KUKA KRL program: ho_60101.src, ho_60101.dat

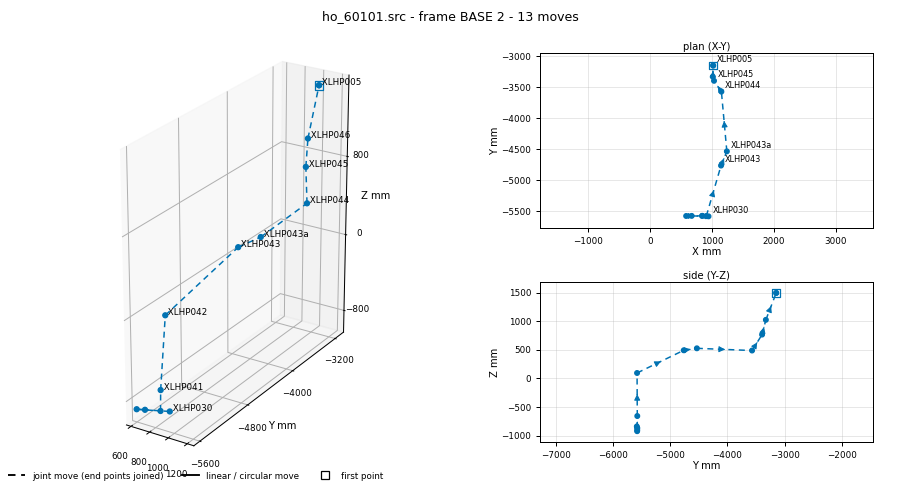
[picture p0: tool path of ho_60101.src in frame BASE 2, 13 of 19 moves have a stored position in this frame; points joined in program order, loops and branches not executed]
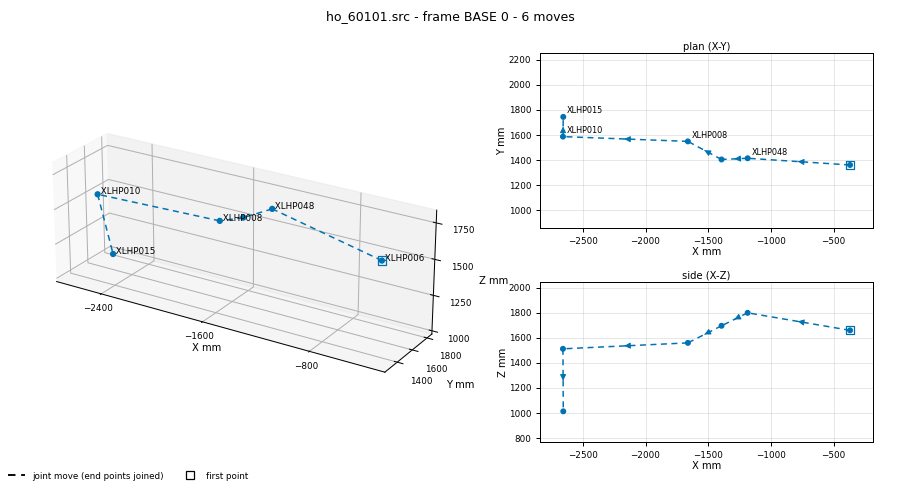
[picture p1: tool path of ho_60101.src in frame BASE 0, 6 of 19 moves have a stored position in this frame; points joined in program order, loops and branches not executed]
--- ho_60101.src ---
&ACCESS RVO2
&REL 599
&COMMENT Pega Lateral
&PARAM DISKPATH = KRC:\R1\Program\MANIPULACAO LTC
DEF ho_60101( )
;FOLD INI
   ;FOLD BASISTECH INI
      GLOBAL INTERRUPT DECL 3 WHEN $STOPMESS==TRUE DO IR_STOPM ( )
      INTERRUPT ON 3
      BAS (#INITMOV,0 )
   ;ENDFOLD (BASISTECH INI)
   ;FOLD SPOTTECH INI
      USERSPOT(#INIT)
   ;ENDFOLD (SPOTTECH INI)
   ;FOLD GRIPPERTECH INI
      USER_GRP(0,DUMMY,DUMMY,GDEFAULT)
   ;ENDFOLD (GRIPPERTECH INI)
   ;FOLD USER INI
      ;Make your modifications here

   ;ENDFOLD (USER INI)
;ENDFOLD (INI)

; Estacao P13.060 - Robo R1
; Programa: Pega da Lateral Accelo (GRIPPER)
; Caracterização dos meios de produção:
; 02/09/2014 09:15 Changes by KUKA Roboter do Brasil

chk_w2_wechs_ok ( )           ; CHECK FERRAMENTA: GRIPPER

;FOLD Kollision.Ueberwachung_3_Ein ;%{PE}%MKUKATPUSER
COLLSTOP( 3, 1 ) ;INTERRUPTUEBERWACHT
;ENDFOLD

;FOLD PTP LHP005  Vel=50 % PDAT23 Tool[2] Base[2];%{PE}%R 4.1.15,%MKUKATPBASIS,%CMOVE,%VPTP,%P 1:PTP, 2:LHP005, 3:, 5:50, 7:PDAT23
$BWDSTART=FALSE
PDAT_ACT=PPDAT23
BAS (#PTP_DAT )
FDAT_ACT=FLHP005
BAS (#FRAMES )
BAS (#VEL_PTP,50 )
PTP  XLHP005
;ENDFOLD
;FOLD PTP LHP006 Vel=100 % PDAT1 Tool[2]:Gripper Lat Esq Accelo Base[0];%{PE}%R 8.2.20,%MKUKATPBASIS,%CMOVE,%VPTP,%P 1:PTP, 2:LHP006, 3:, 5:100, 7:PDAT1
$BWDSTART=FALSE
PDAT_ACT=PPDAT1
FDAT_ACT=FLHP006
BAS(#PTP_PARAMS,100)
PTP XLHP006
;ENDFOLD

;FOLD SET GRP 1  State= OPN  GDAT7;%{PE}%R 4.1.7,%MKUKATPGRP,%CGRP,%VGRP,%P 2:1, 4:1, 5:#NO, 6:GDAT7, 8:0, 10:0
H50(GRP,1,1,GGDAT7)
;ENDFOLD
chk_grp1_opn ( )

;FOLD OUT 3351 'R1_Busca Peca Accelo' State=TRUE ;%{PE}%R 8.2.20,%MKUKATPBASIS,%COUT,%VOUTX,%P 2:3351, 3:R1_Busca Peca Accelo, 5:TRUE, 6:
$OUT[3351]=TRUE
;ENDFOLD
;FOLD OUT 3361 'R1_Solicita Lib. Entrar EST 060EL_621' State=TRUE ;%{PE}%R 8.2.20,%MKUKATPBASIS,%COUT,%VOUTX,%P 2:3361, 3:R1_Solicita Lib. Entrar EST 060EL_621, 5:TRUE, 6:
$OUT[3361]=TRUE
;ENDFOLD
;FOLD WAIT FOR ( IN 3351 'R1_Aguarda Lib. Buscar Lat. Accelo' );%{PE}%R 8.2.20,%MKUKATPBASIS,%CEXT_WAIT_FOR,%VEXT_WAIT_FOR,%P 2:, 4:, 5:$IN, 6:3351, 7:R1_Aguarda Lib. Buscar Lat. Accelo, 9:
WAIT FOR  ( $IN[3351] )
;ENDFOLD
;FOLD OUT 3351 'R1_Busca Peca Accelo' State=FALSE ;%{PE}%R 8.2.20,%MKUKATPBASIS,%COUT,%VOUTX,%P 2:3351, 3:R1_Busca Peca Accelo, 5:FALSE, 6:
$OUT[3351]=FALSE
;ENDFOLD
;FOLD OUT 3361 'R1_Solicita Lib. Entrar EST 060EL_621' State=FALSE ;%{PE}%R 8.2.20,%MKUKATPBASIS,%COUT,%VOUTX,%P 2:3361, 3:R1_Solicita Lib. Entrar EST 060EL_621, 5:FALSE, 6:
$OUT[3361]=FALSE
;ENDFOLD
;FOLD OUT 3367 'R1_Solda Respot Geo1 OK' State=FALSE ;%{PE}%R 8.2.20,%MKUKATPBASIS,%COUT,%VOUTX,%P 2:3367, 3:R1_Solda Respot Geo1 OK, 5:FALSE, 6:
$OUT[3367]=FALSE
;ENDFOLD

;FOLD PTP LHP048 CONT Vel=100 % PDAT12 Tool[2]:Gripper Lat Esq Accelo Base[0];%{PE}%R 8.2.20,%MKUKATPBASIS,%CMOVE,%VPTP,%P 1:PTP, 2:LHP048, 3:C_DIS, 5:100, 7:PDAT12
$BWDSTART=FALSE
PDAT_ACT=PPDAT12
FDAT_ACT=FLHP048
BAS(#PTP_PARAMS,100)
PTP XLHP048 C_DIS
;ENDFOLD
;FOLD PTP LHP007 CONT Vel=100 % PDAT11 Tool[2]:Gripper Lat Esq Accelo Base[0];%{PE}%R 8.2.20,%MKUKATPBASIS,%CMOVE,%VPTP,%P 1:PTP, 2:LHP007, 3:C_DIS, 5:100, 7:PDAT11
$BWDSTART=FALSE
PDAT_ACT=PPDAT11
FDAT_ACT=FLHP007
BAS(#PTP_PARAMS,100)
PTP XLHP007 C_DIS
;ENDFOLD
;FOLD PTP LHP008 CONT Vel=100 % PDAT13 Tool[2]:Gripper Lat Esq Accelo Base[0];%{PE}%R 8.2.20,%MKUKATPBASIS,%CMOVE,%VPTP,%P 1:PTP, 2:LHP008, 3:C_DIS, 5:100, 7:PDAT13
$BWDSTART=FALSE
PDAT_ACT=PPDAT13
FDAT_ACT=FLHP008
BAS(#PTP_PARAMS,100)
PTP XLHP008 C_DIS
;ENDFOLD
;FOLD PTP LHP010 CONT Vel=100 % PDAT14 Tool[2]:Gripper Lat Esq Accelo Base[0];%{PE}%R 8.2.20,%MKUKATPBASIS,%CMOVE,%VPTP,%P 1:PTP, 2:LHP010, 3:C_DIS, 5:100, 7:PDAT14
$BWDSTART=FALSE
PDAT_ACT=PPDAT14
FDAT_ACT=FLHP010
BAS(#PTP_PARAMS,100)
PTP XLHP010 C_DIS
;ENDFOLD
;FOLD PTP LHP015 CONT Vel= 80 % PDAT17 Tool[2]:Gripper Lat Esq Accelo Base[0];%{PE}%R 4.1.16,%MKUKATPBASIS,%CMOVE,%VPTP,%P 1:PTP, 2:LHP015, 3:C_PTP, 5:80, 7:PDAT17
$BWDSTART = FALSE
PDAT_ACT=PPDAT17
BAS(#PTP_DAT)
FDAT_ACT=FLHP015
BAS(#FRAMES)
BAS(#VEL_PTP,80)
PTP XLHP015 C_PTP
;ENDFOLD
;FOLD PTP LHP030 CONT Vel= 50 % PDAT2 Tool[2]:Gripper Lat Esq Accelo Base[0];%{PE}%R 4.1.16,%MKUKATPBASIS,%CMOVE,%VPTP,%P 1:PTP, 2:LHP030, 3:C_PTP, 5:50, 7:PDAT2
$BWDSTART = FALSE
PDAT_ACT=PPDAT2
BAS(#PTP_DAT)
FDAT_ACT=FLHP030
BAS(#FRAMES)
BAS(#VEL_PTP,50)
PTP XLHP030 C_PTP
;ENDFOLD

;FOLD OUT 3386 'Area do Operador (INTERLOCK RB15)' State=FALSE ;%{PE}%R 8.2.20,%MKUKATPBASIS,%COUT,%VOUTX,%P 2:3386, 3:Area do Operador (INTERLOCK RB15), 5:FALSE, 6:
$OUT[3386]=FALSE
;ENDFOLD

;FOLD PTP LHP035 CONT Vel= 50 % PDAT22 Tool[2]:Gripper Lat Esq Accelo Base[0];%{PE}%R 4.1.16,%MKUKATPBASIS,%CMOVE,%VPTP,%P 1:PTP, 2:LHP035, 3:C_PTP, 5:50, 7:PDAT22
$BWDSTART = FALSE
PDAT_ACT=PPDAT22
BAS(#PTP_DAT)
FDAT_ACT=FLHP035
BAS(#FRAMES)
BAS(#VEL_PTP,50)
PTP XLHP035 C_PTP
;ENDFOLD

;FOLD ; posicao de pega;%{PE}%R2.2,%MKUKATPBASIS,%CCOMMENT,%VNORMAL,%P 2: posicao de pega
;ENDFOLD
;FOLD LIN Pick_pos  Vel=2.0 m/s CPDAT1 Tool[2] Base[2];%{PE}%R 4.1.15,%MKUKATPBASIS,%CMOVE,%VLIN,%P 1:LIN, 2:Pick_pos, 3:, 5:2.0, 7:CPDAT1
$BWDSTART=FALSE
LDAT_ACT=LCPDAT1
BAS(#CP_DAT )
FDAT_ACT=FPick_pos
BAS(#FRAMES )
BAS(#VEL_CP,2.0 )
LIN  XPick_pos
;ENDFOLD
;
IF (NOT(GHOST())) then
;FOLD WAIT FOR IN 1 'Presenca de peca gripper'  State= TRUE ;%{PE}%R 4.1.16,%MKUKATPBASIS,%CWAIT_FOR,%VWAIT_FOR,%P 1:0, 2:1, 3:'Presenca de peca gripper', 5:TRUE, 6:
WAIT FOR $IN[1]==TRUE
;ENDFOLD
ENDIF

;FOLD SET GRP 1  State= CLO  GDAT2;%{PE}%R 4.1.7,%MKUKATPGRP,%CGRP,%VGRP,%P 2:1, 4:2, 5:#NO, 6:GDAT2, 8:0, 10:0
H50(GRP,1,2,GGDAT2)
;ENDFOLD
chk_grp1_clo ( )

IF (NOT(GHOST())) then
;FOLD SET GRP 3  State= VACUUM  GDAT3;%{PE}%R 4.1.7,%MKUKATPGRP,%CGRP,%VGRP,%P 2:3, 4:1, 5:#NO, 6:GDAT3, 8:0, 10:0
H50(GRP,3,1,GGDAT3)
;ENDFOLD
;FOLD WAIT FOR ( IN 5 'Vacuo OK' );%{PE}%R 8.2.20,%MKUKATPBASIS,%CEXT_WAIT_FOR,%VEXT_WAIT_FOR,%P 2:, 4:, 5:$IN, 6:5, 7:Vacuo OK, 9:
WAIT FOR  ( $IN[5] )
;ENDFOLD
ENDIF


; Espera sinal plc para sair
;FOLD OUT 3350 'R1_Solicita Lib. Sair Magazine' State=TRUE ;%{PE}%R 8.2.20,%MKUKATPBASIS,%COUT,%VOUTX,%P 2:3350, 3:R1_Solicita Lib. Sair Magazine, 5:TRUE, 6:
$OUT[3350]=TRUE
;ENDFOLD
;FOLD WAIT FOR ( IN 3349 'R1_Aguarda Lib. Sair Magazine' );%{PE}%R 8.2.20,%MKUKATPBASIS,%CEXT_WAIT_FOR,%VEXT_WAIT_FOR,%P 2:, 4:, 5:$IN, 6:3349, 7:R1_Aguarda Lib. Sair Magazine, 9:
WAIT FOR  ( $IN[3349] )
;ENDFOLD
;FOLD OUT 3350 'R1_Solicita Lib. Sair Magazine' State=FALSE ;%{PE}%R 8.2.20,%MKUKATPBASIS,%COUT,%VOUTX,%P 2:3350, 3:R1_Solicita Lib. Sair Magazine, 5:FALSE, 6:
$OUT[3350]=FALSE
;ENDFOLD

;  posicao segura para sair
;FOLD PTP LHP040  Vel= 80 % PDAT3 Tool[2]:Gripper Lat  Esq Accelo Base[2]:Accelo;%{PE}%R 4.1.16,%MKUKATPBASIS,%CMOVE,%VPTP,%P 1:PTP, 2:LHP040, 3:, 5:80, 7:PDAT3
$BWDSTART = FALSE
PDAT_ACT=PPDAT3
BAS(#PTP_DAT)
FDAT_ACT=FLHP040
BAS(#FRAMES)
BAS(#VEL_PTP,80)
PTP XLHP040
;ENDFOLD
;FOLD PTP LHP041 CONT Vel=50 % PDAT4 Tool[2]:Gripper Lat Esq Accelo Base[0];%{PE}%R 8.2.20,%MKUKATPBASIS,%CMOVE,%VPTP,%P 1:PTP, 2:LHP041, 3:C_DIS, 5:50, 7:PDAT4
$BWDSTART=FALSE
PDAT_ACT=PPDAT4
FDAT_ACT=FLHP041
BAS(#PTP_PARAMS,50)
PTP XLHP041 C_DIS
;ENDFOLD
;FOLD PTP LHP042 CONT Vel=50 % PDAT5 Tool[2]:Gripper Lat Esq Accelo Base[0];%{PE}%R 8.2.20,%MKUKATPBASIS,%CMOVE,%VPTP,%P 1:PTP, 2:LHP042, 3:C_DIS, 5:50, 7:PDAT5
$BWDSTART=FALSE
PDAT_ACT=PPDAT5
FDAT_ACT=FLHP042
BAS(#PTP_PARAMS,50)
PTP XLHP042 C_DIS
;ENDFOLD
;FOLD PTP LHP043 CONT Vel=50 % PDAT6 Tool[2]:Gripper Lat Esq Accelo Base[0];%{PE}%R 8.2.20,%MKUKATPBASIS,%CMOVE,%VPTP,%P 1:PTP, 2:LHP043, 3:C_DIS, 5:50, 7:PDAT6
$BWDSTART=FALSE
PDAT_ACT=PPDAT6
FDAT_ACT=FLHP043
BAS(#PTP_PARAMS,50)
PTP XLHP043 C_DIS
;ENDFOLD
;FOLD PTP LHP043a CONT Vel=50 % PDAT8 Tool[2]:Gripper Lat Esq Accelo Base[0];%{PE}%R 8.2.20,%MKUKATPBASIS,%CMOVE,%VPTP,%P 1:PTP, 2:LHP043a, 3:C_DIS, 5:50, 7:PDAT8
$BWDSTART=FALSE
PDAT_ACT=PPDAT8
FDAT_ACT=FLHP043a
BAS(#PTP_PARAMS,50)
PTP XLHP043a C_DIS
;ENDFOLD
;FOLD PTP LHP044 CONT Vel=50 % PDAT7 Tool[2]:Gripper Lat Esq Accelo Base[0];%{PE}%R 8.2.20,%MKUKATPBASIS,%CMOVE,%VPTP,%P 1:PTP, 2:LHP044, 3:C_DIS, 5:50, 7:PDAT7
$BWDSTART=FALSE
PDAT_ACT=PPDAT7
FDAT_ACT=FLHP044
BAS(#PTP_PARAMS,50)
PTP XLHP044 C_DIS
;ENDFOLD

;FOLD OUT 3386 'Area do Operador (INTERLOCK RB15)' State=TRUE ;%{PE}%R 8.2.20,%MKUKATPBASIS,%COUT,%VOUTX,%P 2:3386, 3:Area do Operador (INTERLOCK RB15), 5:TRUE, 6:
$OUT[3386]=TRUE
;ENDFOLD

;FOLD PTP LHP045 CONT Vel= 80 % P_OLP6 Tool[2]:Gripper Lat Esq Accelo Base[0];%{PE}%R 4.1.16,%MKUKATPBASIS,%CMOVE,%VPTP,%P 1:PTP, 2:LHP045, 3:C_PTP, 5:80, 7:P_OLP6
$BWDSTART = FALSE
PDAT_ACT=PP_OLP6
BAS(#PTP_DAT)
FDAT_ACT=FLHP045
BAS(#FRAMES)
BAS(#VEL_PTP,80)
PTP XLHP045 C_PTP
;ENDFOLD
;FOLD PTP LHP046 CONT Vel=50 % PDAT9 Tool[2]:Gripper Lat Esq Accelo Base[0];%{PE}%R 8.2.20,%MKUKATPBASIS,%CMOVE,%VPTP,%P 1:PTP, 2:LHP046, 3:C_DIS, 5:50, 7:PDAT9
$BWDSTART=FALSE
PDAT_ACT=PPDAT9
FDAT_ACT=FLHP046
BAS(#PTP_PARAMS,50)
PTP XLHP046 C_DIS
;ENDFOLD
;FOLD PTP LHP075  Vel= 80 % PDAT24 Tool[2]:Gripper Lat  Esq Accelo Base[2]:Accelo;%{PE}%R 4.1.16,%MKUKATPBASIS,%CMOVE,%VPTP,%P 1:PTP, 2:LHP075, 3:, 5:80, 7:PDAT24
$BWDSTART = FALSE
PDAT_ACT=PPDAT24
BAS(#PTP_DAT)
FDAT_ACT=FLHP075
BAS(#FRAMES)
BAS(#VEL_PTP,80)
PTP XLHP075
;ENDFOLD

;FOLD OUT 3351 'R1_Busca Peca Accelo' State=TRUE ;%{PE}%R 8.2.20,%MKUKATPBASIS,%COUT,%VOUTX,%P 2:3351, 3:R1_Busca Peca Accelo, 5:TRUE, 6:
$OUT[3351]=TRUE
;ENDFOLD
;FOLD PULSE 3349 'R1_Pegou Peca' State=TRUE Time=3 sec;%{PE}%R 8.2.20,%MKUKATPBASIS,%COUT,%VPULSE,%P 2:3349, 3:R1_Pegou Peca, 5:TRUE, 6:, 8:3
PULSE($OUT[3349], TRUE,3)
;ENDFOLD

END

--- ho_60101.dat ---
&ACCESS RVO2
&REL 599
&COMMENT Pega Lateral
&PARAM DISKPATH = KRC:\R1\Program\MANIPULACAO LTC
DEFDAT  ho_60101
;FOLD EXTERNAL DECLARATIONS;%{PE}%MKUKATPBASIS,%CEXT,%VCOMMON,%P
;FOLD GRIPPERTECH EXT
EXT  H50 (INT  :IN,INT  :IN,INT  :IN,GRP_TYP  :IN )
;ENDFOLD (GRIPPERTECH EXT)
;FOLD SPOTTECH EXT
EXT  USERSPOT (S_COMMAND  :IN,SPOT_TYPE  :IN )
;ENDFOLD (SPOTTECH EXT)
;FOLD BASISTECH EXT;%{PE}%MKUKATPBASIS,%CEXT,%VEXT,%P
EXT  BAS (BAS_COMMAND  :IN,REAL  :IN )
DECL INT SUCCESS
;ENDFOLD (BASISTECH EXT)
;FOLD USER EXT;%{E}%MKUKATPUSER,%CEXT,%VEXT,%P
;Make your modifications here

;ENDFOLD (USER EXT)
;ENDFOLD (EXTERNAL DECLARATIONS)

;# ============ START PATH : bh_p13060r1_ltc_01 =============
DECL FDAT FLHP040={TOOL_NO 2,BASE_NO 2,IPO_FRAME #BASE}
DECL E6POS XLHP040={X 838.254578,Y -5574.66309,Z -866.243774,A 89.6557083,B 0.696913004,C -102.786201,S 18,T 35,E1 0.0,E2 0.0,E3 0.0,E4 0.0,E5 0.0,E6 0.0}
DECL FDAT FLHP045={TOOL_NO 2,BASE_NO 2,IPO_FRAME #BASE}
DECL PDAT PP_OLP6={VEL 100.0,ACC 100.0,APO_DIST 100.0}
DECL E6POS XLHP045={X 1031.34094,Y -3395.22192,Z 766.315613,A 82.4350967,B -0.70792228,C -83.1183472,S 18,T 35,E1 0.0,E2 0.0,E3 0.0,E4 0.0,E5 0.0,E6 0.0}
DECL E6POS XLHP030={X 942.53479,Y -5582.48291,Z -837.87439,A 89.7051163,B 0.529519916,C -102.831596,S 2,T 35,E1 0.0,E2 0.0,E3 0.0,E4 0.0,E5 0.0,E6 0.0}
DECL FDAT FLHP030={TOOL_NO 2,BASE_NO 2,IPO_FRAME #BASE}
DECL PDAT PPDAT2={VEL 100.0,ACC 100.0,APO_DIST 5.0}
DECL PDAT PPDAT3={VEL 100.0,ACC 100.0,APO_DIST 100.0}
DECL GRP_SUGG_T LAST_GRP={NUMBER[] "1                       ",STATE[] "1                       ",PARAMS[] "GDAT7                   "}
DECL GRP_TYP GGDAT1={G_APO #NO,GRP_TIME 0.200000003,CTRL #OFF,DLY 0,DST 1}
DECL GRP_TYP GGDAT2={G_APO #NO,GRP_TIME 0.200000003,CTRL #OFF,DLY 0,DST 1}
DECL GRP_TYP GGDAT3={G_APO #NO,GRP_TIME 0.200000003,CTRL #OFF,DLY 0,DST 1}
DECL GRP_TYP GGDAT4={G_APO #NO,GRP_TIME 0.200000003,CTRL #OFF,DLY 0,DST 1}
DECL GRP_TYP GGDAT5={G_APO #NO,GRP_TIME 0.200000003,CTRL #OFF,DLY 0,DST 1}
DECL E6POS XLHP010={X -2658.55298,Y 1587.45496,Z 1512.15198,A -2.75169802,B 1.47639501,C -107.936096,S 18,T 35,E1 0.0,E2 0.0,E3 0.0,E4 0.0,E5 0.0,E6 0.0}
DECL FDAT FLHP010={TOOL_NO 2,BASE_NO 0,IPO_FRAME #BASE}
DECL E6POS XLHP015={X -2656.13208,Y 1744.65796,Z 1013.55701,A -2.75470901,B 1.48318195,C -108.002502,S 18,T 35,E1 0.0,E2 0.0,E3 0.0,E4 0.0,E5 0.0,E6 0.0}
DECL FDAT FLHP015={TOOL_NO 2,BASE_NO 0,IPO_FRAME #BASE}
DECL PDAT PPDAT17={VEL 100.0,ACC 100.0,APO_DIST 100.0}
DECL GRP_TYP GGDAT6={G_APO #NO,GRP_TIME 0.200000003,CTRL #OFF,DLY 0,DST 1}
DECL GRP_TYP GGDAT7={G_APO #NO,GRP_TIME 0.200000003,CTRL #OFF,DLY 0,DST 1}
DECL E6POS XLHP035={X 670.721191,Y -5574.84619,Z -901.981323,A 89.6396027,B 0.701093078,C -103.174599,S 18,T 35,E1 0.0,E2 0.0,E3 0.0,E4 0.0,E5 0.0,E6 0.0}
DECL FDAT FLHP035={TOOL_NO 2,BASE_NO 2,IPO_FRAME #BASE}
DECL PDAT PPDAT22={VEL 100.0,ACC 100.0,APO_DIST 5.0}
DECL PDAT PPDAT23={VEL 50.0,ACC 100.0,APO_DIST 10.0}
DECL E6POS XLHP075={X 1017.82898,Y -3148.71802,Z 1493.39404,A 4.49403811,B 78.8011627,C -170.569595,S 2,T 35,E1 0.0,E2 0.0,E3 0.0,E4 0.0,E5 0.0,E6 0.0}
DECL FDAT FLHP075={TOOL_NO 2,BASE_NO 2,IPO_FRAME #BASE}
DECL PDAT PPDAT24={VEL 100.0,ACC 100.0,APO_DIST 10.0}
DECL LDAT LCPDAT1={VEL 2.0,ACC 100.0,APO_DIST 100.0,APO_FAC 50.0}
DECL E6POS XPick_pos={X 581.659302,Y -5576.59277,Z -920.624817,A 89.7079163,B 1.09576297,C -102.428299,S 18,T 35,E1 0.0,E2 0.0,E3 0.0,E4 0.0,E5 0.0,E6 0.0}
DECL FDAT FPick_pos={TOOL_NO 2,BASE_NO 2,IPO_FRAME #BASE}
DECL E6POS XLHP005={X 1017.82898,Y -3148.71704,Z 1493.39502,A 4.49398613,B 78.8012009,C -170.569595,S 2,T 35,E1 0.0,E2 0.0,E3 0.0,E4 0.0,E5 0.0,E6 0.0}
DECL FDAT FLHP005={TOOL_NO 2,BASE_NO 2,IPO_FRAME #BASE}
DECL BASIS_SUGG_T LAST_BASIS={POINT1[] "LHP048                  ",POINT2[] "LHP048                  ",CP_PARAMS[] "CPDAT4                  ",PTP_PARAMS[] "PDAT12                  ",CONT[] "C_DIS                   ",CP_VEL[] "1                       ",PTP_VEL[] "100                     ",SYNC_PARAMS[] "SYNCDAT                 ",SPL_NAME[] "S0                      "}
DECL E6POS XLHP006={X -368.39151,Y 1361.11304,Z 1659.71802,A -0.79789108,B -0.378875285,C -112.862396,S 18,T 11,E1 0.0,E2 0.0,E3 0.0,E4 0.0,E5 0.0,E6 0.0}
DECL FDAT FLHP006={TOOL_NO 2,BASE_NO 0,IPO_FRAME #BASE,POINT2[] " ",TQ_STATE FALSE}
DECL PDAT PPDAT1={VEL 100.0,ACC 100.0,APO_DIST 100.0,GEAR_JERK 50.0}
DECL LDAT LCPDAT2={VEL 2.0,ACC 50.0,APO_DIST 100.0,APO_FAC 50.0,AXIS_VEL 100.0,AXIS_ACC 100.0,ORI_TYP #VAR,CIRC_TYP #BASE,JERK_FAC 50.0,GEAR_JERK 50.0,EXAX_IGN 0}
DECL E6POS XLHP007={X -1393.56396,Y 1405.05505,Z 1695.875,A -1.87000704,B 0.636861086,C -110.161598,S 18,T 35,E1 0.0,E2 0.0,E3 0.0,E4 0.0,E5 0.0,E6 0.0}
DECL FDAT FLHP007={TOOL_NO 2,BASE_NO 0,IPO_FRAME #BASE,POINT2[] " ",TQ_STATE FALSE}
DECL LDAT LCPDAT3={VEL 2.0,ACC 50.0,APO_DIST 100.0,APO_FAC 50.0,AXIS_VEL 100.0,AXIS_ACC 100.0,ORI_TYP #VAR,CIRC_TYP #BASE,JERK_FAC 50.0,GEAR_JERK 50.0,EXAX_IGN 0}
DECL E6POS XLHP008={X -1661.89697,Y 1549.32605,Z 1559.50305,A -2.13267398,B 0.891956985,C -109.509102,S 18,T 35,E1 0.0,E2 0.0,E3 0.0,E4 0.0,E5 0.0,E6 0.0}
DECL FDAT FLHP008={TOOL_NO 2,BASE_NO 0,IPO_FRAME #BASE,POINT2[] " ",TQ_STATE FALSE}
DECL LDAT LCPDAT4={VEL 2.0,ACC 50.0,APO_DIST 100.0,APO_FAC 50.0,AXIS_VEL 100.0,AXIS_ACC 100.0,ORI_TYP #VAR,CIRC_TYP #BASE,JERK_FAC 50.0,GEAR_JERK 50.0,EXAX_IGN 0}
DECL E6POS XLHP041={X 842.897827,Y -5574.10889,Z -655.778625,A 89.3989334,B -13.9881802,C -99.0561829,S 18,T 35,E1 0.0,E2 0.0,E3 0.0,E4 0.0,E5 0.0,E6 0.0}
DECL FDAT FLHP041={TOOL_NO 2,BASE_NO 2,IPO_FRAME #BASE,POINT2[] " ",TQ_STATE FALSE}
DECL PDAT PPDAT4={VEL 100.0,ACC 100.0,APO_DIST 100.0,APO_MODE #CDIS,GEAR_JERK 50.0}
DECL E6POS XLHP042={X 906.871277,Y -5577.9292,Z 95.8650284,A 88.6567383,B -2.11703706,C -92.0317688,S 18,T 35,E1 0.0,E2 0.0,E3 0.0,E4 0.0,E5 0.0,E6 0.0}
DECL FDAT FLHP042={TOOL_NO 2,BASE_NO 2,IPO_FRAME #BASE,POINT2[] " ",TQ_STATE FALSE}
DECL PDAT PPDAT5={VEL 100.0,ACC 100.0,APO_DIST 100.0,APO_MODE #CDIS,GEAR_JERK 50.0}
DECL E6POS XLHP043={X 1144.5,Y -4762.86719,Z 491.821686,A 88.659668,B -2.11881399,C -92.0398865,S 18,T 35,E1 0.0,E2 0.0,E3 0.0,E4 0.0,E5 0.0,E6 0.0}
DECL FDAT FLHP043={TOOL_NO 2,BASE_NO 2,IPO_FRAME #BASE,POINT2[] " ",TQ_STATE FALSE}
DECL PDAT PPDAT6={VEL 100.0,ACC 100.0,APO_DIST 100.0,APO_MODE #CDIS,GEAR_JERK 50.0}
DECL E6POS XLHP044={X 1150.29895,Y -3570.01807,Z 487.99411,A 88.6528091,B -2.07348609,C -92.0989532,S 18,T 35,E1 0.0,E2 0.0,E3 0.0,E4 0.0,E5 0.0,E6 0.0}
DECL FDAT FLHP044={TOOL_NO 2,BASE_NO 2,IPO_FRAME #BASE,POINT2[] " ",TQ_STATE FALSE}
DECL PDAT PPDAT7={VEL 100.0,ACC 100.0,APO_DIST 100.0,APO_MODE #CDIS,GEAR_JERK 50.0}
DECL E6POS XLHP043A={X 1238.22302,Y -4533.76221,Z 526.550171,A 88.7746582,B -1.41036403,C -91.4281235,S 18,T 35,E1 0.0,E2 0.0,E3 0.0,E4 0.0,E5 0.0,E6 0.0}
DECL FDAT FLHP043a={TOOL_NO 2,BASE_NO 2,IPO_FRAME #BASE,POINT2[] " ",TQ_STATE FALSE}
DECL PDAT PPDAT8={VEL 100.0,ACC 100.0,APO_DIST 100.0,APO_MODE #CDIS,GEAR_JERK 50.0}
DECL E6POS XLHP046={X 1011.28198,Y -3329.18994,Z 1023.70502,A 78.8528366,B 27.6525898,C -87.816452,S 18,T 35,E1 0.0,E2 0.0,E3 0.0,E4 0.0,E5 0.0,E6 0.0}
DECL FDAT FLHP046={TOOL_NO 2,BASE_NO 2,IPO_FRAME #BASE,POINT2[] " ",TQ_STATE FALSE}
DECL PDAT PPDAT9={VEL 100.0,ACC 100.0,APO_DIST 100.0,APO_MODE #CDIS,GEAR_JERK 50.0}
DECL PDAT PPDAT11={VEL 100.0,ACC 100.0,APO_DIST 15.0,APO_MODE #CDIS,GEAR_JERK 50.0}
DECL E6POS XLHP048={X -1185.21997,Y 1414.68799,Z 1799.43298,A -2.28385901,B -1.065395,C -115.208,S 18,T 35,E1 0.0,E2 0.0,E3 0.0,E4 0.0,E5 0.0,E6 0.0}
DECL FDAT FLHP048={TOOL_NO 2,BASE_NO 0,IPO_FRAME #BASE,POINT2[] " ",TQ_STATE FALSE}
DECL PDAT PPDAT12={VEL 100.0,ACC 100.0,APO_DIST 15.0,APO_MODE #CDIS,GEAR_JERK 50.0}
DECL PDAT PPDAT13={VEL 100.0,ACC 100.0,APO_DIST 15.0,APO_MODE #CDIS,GEAR_JERK 50.0}
DECL PDAT PPDAT14={VEL 100.0,ACC 100.0,APO_DIST 15.0,APO_MODE #CDIS,GEAR_JERK 50.0}
ENDDAT
